FUNCTION_BLOCK F_DAY_OF_WEEK (* get day of week from date *)
  (* Standard: 61131-3; Classification: standard character and string function; Description: Copyright (c) 2013 TU Wien ACIN and others. This program and the accompanying materials are made available under the terms of the Eclipse Public License 2.0 which is available at https://www.eclipse.org/legal/epl-2.0/ SPDX-License-Identifier: EPL-2.0 Some portions generated by Gemini CLI *)
  (* Version 1.0, 2026-01-31, Franz Höpfinger, HR Agrartechnik GmbH, F_CONCAT_TOD copied from an existing fB and implemented according IEC 61131-3 *)
  PACKAGE iec61131::charString;
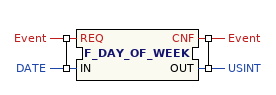
  EVENT_INPUT
    REQ WITH IN; (* Service Request *)
  END_EVENT
  EVENT_OUTPUT
    CNF WITH OUT; (* Confirmation of Requested Service *)
  END_EVENT
  VAR_INPUT
    IN : DATE; (* Input DATE *)
  END_VAR
  VAR_OUTPUT
    OUT : USINT; (* Day of week (0=Sunday, ..., 6=Saturday) *)
  END_VAR
  EC_STATES
    REQ : REQ -> CNF;
  END_STATES
  ALGORITHM REQ IN ST:
OUT := DAY_OF_WEEK(IN);
  END_ALGORITHM
END_FUNCTION_BLOCK
